FUNCTION_BLOCK Integrator
VAR_INPUT
END_VAR
VAR_OUTPUT
END_VAR
VAR
END_VAR

END_FUNCTION_BLOCK

(* stored: Version 1.1.0.1, ProductVersion 3.1.4022.12
   POU Integrator: Id {7444c4be-3c1a-431c-a15f-d1788f7f37e2}, SpecialFunc None *)
